(* CODESYS project GeradorPulso2TPs.project

Project tree, tasks and I/O mapping:
  Device : CODESYS Control Win V3, 3S - Smart Software Solutions GmbH, order no. 305021, version 3.5.11.30
    application Application
      libraries: Standard, * (System)
      task MainTask (cyclic, interval t#20ms, priority 1) calls PLC_PRG
      task VISU_TASK (cyclic, interval 100 ms, priority 31) calls VisuElems.Visu_Prg
      program PLC_PRG [LD]
      visualisation Visualization
  libraries: VisuSymbols, 3.5.10.0 (System)
  text list GlobalTextList
*)

// Device/Application/PLC_PRG
PROGRAM PLC_PRG
VAR
	Start : BOOL;
	Stop : BOOL;
	Ton: BOOL;
	Pulsos_IN: BOOL;
	Tempo_Operacao : BOOL;
	
	TP_1 : TP;
	ET_1 : TIME;
	
	TP_2: TP;
	ET_2 : TIME;
END_VAR
VAR // added by the converter: edge detectors and wires of the graphical bodies
    _rt1 : R_TRIG;
    _ft1, _ft2 : F_TRIG;
END_VAR

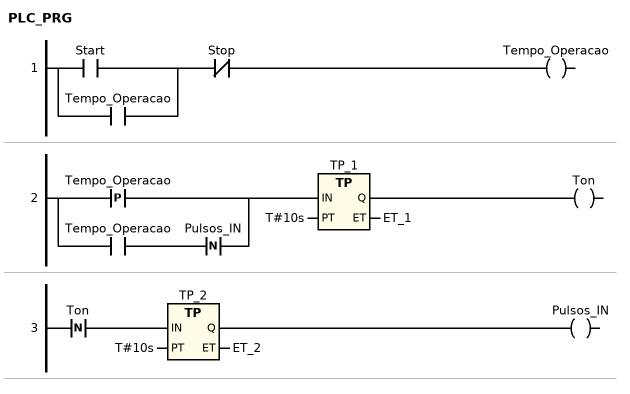
// NETWORK 1
Tempo_Operacao := (Start OR Tempo_Operacao) AND NOT Stop;

// NETWORK 2
_rt1(CLK := Tempo_Operacao);
_ft1(CLK := Pulsos_IN);
TP_1(IN := _rt1.Q OR Tempo_Operacao AND _ft1.Q, PT := T#10s, ET => ET_1); // TP
Ton := TP_1.Q;

// NETWORK 3
_ft2(CLK := Ton);
TP_2(IN := _ft2.Q, PT := T#10s, ET => ET_2); // TP
Pulsos_IN := TP_2.Q;

END_PROGRAM

// Device/Application/Visualization
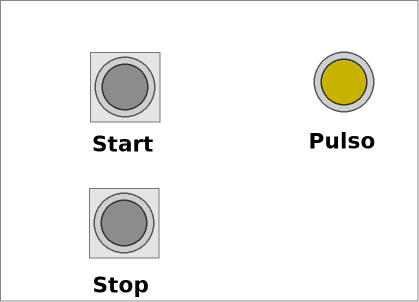
VISUALIZATION Visualization  // 419x302
    PushSwitchLed (90,52 70x70), variable: PLC_PRG.Start, behaviour: TOGGLE, style: Switch-PushSwitchLed-Gray
    PushSwitchLed (89,188 70x70), variable: PLC_PRG.Stop, behaviour: TOGGLE, style: Switch-PushSwitchLed-Gray
    Lamp1 (309,47 70x70), variable: PLC_PRG.Pulsos_IN, style: Lamp-Lamp1-Yellow
    Label (48,129 150x30), "Start"
    Label (267,126 150x30), "Pulso"
    Label (46,270 150x30), "Stop"
END_VISUALIZATION
